gfCNCPoint2[29961] = {X 20.0868, Y 58.7965, Z -3.8333, A 0.000, B 0.000, C 0.000 }
gfCNCPoint2[29962] = {X 17.4734, Y 59.3123, Z -3.8333, A 0.000, B 0.000, C 0.000 }
gfCNCPoint2[29963] = {X 14.8265, Y 59.6126, Z -3.8333, A 0.000, B 0.000, C 0.000 }
gfCNCPoint2[29964] = {X 12.1639, Y 59.6953, Z -3.8333, A 0.000, B 0.000, C 0.000 }
gfCNCPoint2[29965] = {X 9.5035, Y 59.5598, Z -3.8333, A 0.000, B 0.000, C 0.000 }
gfCNCPoint2[29966] = {X 9.5035, Y 90.4950, Z -3.8333, A 0.000, B 0.000, C 0.000 }
gfCNCPoint2[29967] = {X 114.8629, Y 90.4950, Z -3.8333, A 0.000, B 0.000, C 0.000 }
gfCNCPoint2[29968] = {X 115.7474, Y 89.2983, Z -3.8333, A 0.000, B 0.000, C 0.000 }
gfCNCPoint2[29969] = {X 116.7722, Y 88.2194, Z -3.8333, A 0.000, B 0.000, C 0.000 }
gfCNCPoint2[29970] = {X 117.9220, Y 87.2746, Z -3.8333, A 0.000, B 0.000, C 0.000 }
gfCNCPoint2[29971] = {X 119.1792, Y 86.4785, Z -3.8333, A 0.000, B 0.000, C 0.000 }
gfCNCPoint2[29972] = {X 120.5247, Y 85.8429, Z -3.8333, A 0.000, B 0.000, C 0.000 }
gfCNCPoint2[29973] = {X 121.9381, Y 85.3776, Z -3.8333, A 0.000, B 0.000, C 0.000 }
gfCNCPoint2[29974] = {X 123.3981, Y 85.0896, Z -3.8333, A 0.000, B 0.000, C 0.000 }
gfCNCPoint2[29975] = {X 123.5632, Y 84.9118, Z -3.8333, A 0.000, B 0.000, C 0.000 }
gfCNCPoint2[29976] = {X 123.7264, Y 84.7322, Z -3.8333, A 0.000, B 0.000, C 0.000 }
gfCNCPoint2[29977] = {X 147.2181, Y 58.9351, Z -3.8333, A 0.000, B 0.000, C 0.000 }
gfCNCPoint2[29978] = {X 147.2180, Y 58.0000, Z -3.8333, A 0.000, B 0.000, C 0.000 }
gfCNCPoint2[29979] = {X 147.2987, Y 56.6058, Z -3.8333, A 0.000, B 0.000, C 0.000 }
gfCNCPoint2[29980] = {X 147.5398, Y 55.2303, Z -3.8333, A 0.000, B 0.000, C 0.000 }
gfCNCPoint2[29981] = {X 148.0022, Y 53.7185, Z -3.8333, A 0.000, B 0.000, C 0.000 }
gfCNCPoint2[29982] = {X 148.6580, Y 52.2800, Z -3.8333, A 0.000, B 0.000, C 0.000 }
gfCNCPoint2[29983] = {X 143.0396, Y 52.2800, Z -3.8333, A 0.000, B 0.000, C 0.000 }
gfCNCPoint2[29984] = {X 141.7807, Y 52.1703, Z -3.8333, A 0.000, B 0.000, C 0.000 }
gfCNCPoint2[29985] = {X 140.5597, Y 51.8446, Z -3.8333, A 0.000, B 0.000, C 0.000 }
gfCNCPoint2[29986] = {X 139.4134, Y 51.3126, Z -3.8333, A 0.000, B 0.000, C 0.000 }
gfCNCPoint2[29987] = {X 138.3764, Y 50.5904, Z -3.8333, A 0.000, B 0.000, C 0.000 }
gfCNCPoint2[29988] = {X 137.4799, Y 49.6998, Z -3.8333, A 0.000, B 0.000, C 0.000 }
gfCNCPoint2[29989] = {X 136.7509, Y 48.6675, Z -3.8333, A 0.000, B 0.000, C 0.000 }
gfCNCPoint2[29990] = {X 136.2114, Y 47.5248, Z -3.8333, A 0.000, B 0.000, C 0.000 }
gfCNCPoint2[29991] = {X 135.8777, Y 46.3059, Z -3.8333, A 0.000, B 0.000, C 0.000 }
gfCNCPoint2[29992] = {X 135.7598, Y 45.0477, Z -3.8333, A 0.000, B 0.000, C 0.000 }
gfCNCPoint2[29993] = {X 135.7601, Y 44.1247, Z -3.8333, A 0.000, B 0.000, C 0.000 }
gfCNCPoint2[29994] = {X 135.8408, Y 43.1249, Z -3.8333, A 0.000, B 0.000, C 0.000 }
gfCNCPoint2[29995] = {X 136.0581, Y 42.1457, Z -3.8333, A 0.000, B 0.000, C 0.000 }
gfCNCPoint2[29996] = {X 138.3597, Y 42.8258, Z -3.8333, A 0.000, B 0.000, C 0.000 }
gfCNCPoint2[29997] = {X 138.6721, Y 42.0319, Z -3.8333, A 0.000, B 0.000, C 0.000 }
gfCNCPoint2[29998] = {X 139.1179, Y 41.3046, Z -3.8333, A 0.000, B 0.000, C 0.000 }
gfCNCPoint2[29999] = {X 139.6836, Y 40.6660, Z -3.8333, A 0.000, B 0.000, C 0.000 }
gfCNCPoint2[30000] = {X 139.6836, Y 20.4371, Z -3.8333, A 0.000, B 0.000, C 0.000 }

ENDDAT
